(* PLC project MaterialCartControl, AI-PLC-Integration AI SCL→LAD Generator 1.0 *)
(* stored: creationDateTime 2026-05-30T11:56:26.933728, modificationDateTime 2026-05-30T11:56:26.933728 *)

FUNCTION_BLOCK MaterialCartControl
  VAR_INPUT
    bStart : BOOL;  (* 启动 *)
    bStop : BOOL;  (* 停止 *)
    bReset : BOOL;  (* 复位 *)
    bEmergencyStop : BOOL;  (* 急停（常闭） *)
    bForwardLimit : BOOL;  (* 前限位 *)
    bReverseLimit : BOOL;  (* 后限位 *)
    bOverload : BOOL;  (* 过载（常闭） *)
    bManualMode : BOOL;  (* 手动模式 *)
    bManualForward : BOOL;  (* 手动正转 *)
    bManualReverse : BOOL;  (* 手动反转 *)
  END_VAR
  VAR_OUTPUT
    bForwardOut : BOOL;  (* 正转输出 *)
    bReverseOut : BOOL;  (* 反转输出 *)
    bRunning : BOOL;  (* 运行中 *)
    bFault : BOOL;  (* 故障 *)
  END_VAR
  VAR
    bSafetyOK : BOOL;  (* 安全链正常 *)
    bFaultLatch : BOOL;  (* 故障锁存 *)
    iState1 : BOOL;  (* 状态=前进 *)
    iState2 : BOOL;  (* 状态=卸载 *)
    iState3 : BOOL;  (* 状态=后退 *)
    iState4 : BOOL;  (* 状态=装载 *)
    iState5 : BOOL;  (* 状态=故障 *)
  END_VAR
  VAR_TEMP
    tmrUnload : TON;  (* 卸载延时 T#5S *)
    tmrLoad : TON;  (* 装载延时 T#3S *)
  END_VAR

(* LD diagram, written out as Structured Text *)
END_FUNCTION_BLOCK
